// Mitsubishi GX Works2 project: MOV_word_ops   PLC: Q02/Q02H

PROGRAM MAIN
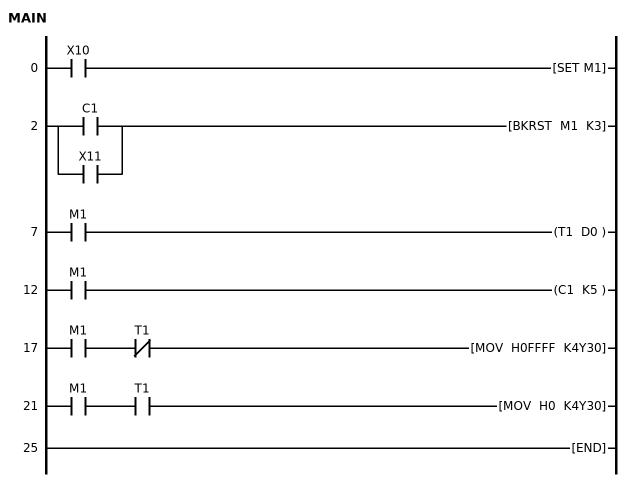
0     LD      X10
      SET     M1
2     LD      C1
      OR      X11
      BKRST   M1 K3
7     LD      M1
      OUT     T1 D0
12    LD      M1
      OUT     C1 K5
17    LD      M1
      ANI     T1
      MOV     H0FFFF K4Y30
21    LD      M1
      AND     T1
      MOV     H0 K4Y30
25    END
END_PROGRAM
